{attribute 'linkalways'} 
{attribute 'no_explicit_call' := 'This FB is a CLASS and must be accessed using methods or properties'}
{attribute 'enable_dynamic_creation'}
FUNCTION_BLOCK _ETcVnKeypointDetectionTypeFAST EXTENDS EnumDatatypeBase
VAR
	localData : ETcVnKeypointDetectionTypeFAST;
	activeData : REFERENCE TO ETcVnKeypointDetectionTypeFAST;
	enumBaseDatatype : _DINT(localData);
END_VAR

METHOD PRIVATE AddLocalEnumeration
VAR_INPUT
	Enumeration : T_MAXSTRING;
	Value : ETcVnKeypointDetectionTypeFAST;
END_VAR
AddEnumeration(Enumeration, Value);
END_METHOD

PROPERTY PUBLIC Address : PVOID
GET
Address := ADR(activeData);
END_GET
END_PROPERTY

METHOD PUBLIC ClearReference
VAR_INPUT
END_VAR
activeData REF= localData;
SetBaseDatatypeReference();
END_METHOD

METHOD PUBLIC Clone : I_Datatype
VAR
    pClone : POINTER TO _ETcVnKeypointDetectionTypeFAST;
END_VAR
pClone := __NEW(_ETcVnKeypointDetectionTypeFAST(InitialValue := Value));
Clone := pClone^;
END_METHOD

METHOD FB_init : BOOL
VAR_INPUT
	bInitRetains : BOOL; // if TRUE, the retain variables are initialized (warm start / cold start)
	bInCopyCode : BOOL;  // if TRUE, the instance afterwards gets moved into the copy code (online change)
	InitialValue : ETcVnKeypointDetectionTypeFAST;
END_VAR
localData := InitialValue;
AddBaseDatatype(enumBaseDatatype);
ClearReference();

AddLocalEnumeration('TCVN_KDT_FAST_5_8', ETcVnKeypointDetectionTypeFAST.TCVN_KDT_FAST_5_8);
AddLocalEnumeration('TCVN_KDT_FAST_7_12', ETcVnKeypointDetectionTypeFAST.TCVN_KDT_FAST_7_12);
AddLocalEnumeration('TCVN_KDT_FAST_9_16', ETcVnKeypointDetectionTypeFAST.TCVN_KDT_FAST_9_16);
END_METHOD

PROPERTY PUBLIC Identifier : T_MAXSTRING
GET
Identifier := 'ETcVnKeypointDetectionTypeFAST';
END_GET
END_PROPERTY

METHOD IsEnumeratorValueEqual : BOOL
VAR_INPUT
	Enumerator : I_KeyValueForwardEnumerator;
END_VAR
VAR
	storedValue : ETcVnKeypointDetectionTypeFAST;
END_VAR
IF NOT Enumerator.TryGet(storedValue) THEN
	RETURN;
END_IF

IsEnumeratorValueEqual := storedValue = activeData;
END_METHOD

METHOD PUBLIC MakeReferenceTo
VAR_INPUT
	ReferenceTarget : REFERENCE TO ETcVnKeypointDetectionTypeFAST;
END_VAR
activeData REF= ReferenceTarget;
SetBaseDatatypeReference();
END_METHOD

METHOD PROTECTED SetBaseDatatypeReference
VAR_INPUT
END_VAR
enumBaseDatatype.MakeReferenceTo(activeData);
END_METHOD

PROPERTY PUBLIC Size : UDINT
GET
Size := SIZEOF(activeData);
END_GET
END_PROPERTY

METHOD TryMakeReferenceTo : BOOL
VAR_INPUT
	Target : I_Datatype;
END_VAR
VAR
	targetAsEnum : I_EnumDatatype;
	pTargetData : POINTER TO ETcVnKeypointDetectionTypeFAST;
END_VAR
IF NOT Target.TryResolveAsEnumDatatype(targetAsEnum) THEN
	RETURN;
END_IF

IF targetAsEnum.Identifier <> Identifier THEN
	RETURN;
END_IF

pTargetData := Target.Address;
activeData REF= pTargetData^;
SetBaseDatatypeReference();
TryMakeReferenceTo := TRUE;
END_METHOD

PROPERTY PUBLIC Value : ETcVnKeypointDetectionTypeFAST
GET
Value := activeData;
END_GET
SET
activeData := Value;
END_SET
END_PROPERTY

END_FUNCTION_BLOCK

(* stored: Version 1.1.0.1, ProductVersion 3.1.4024.12
   POU _ETcVnKeypointDetectionTypeFAST: Id {07be448e-3997-4734-bde9-814ab5e413a9}, SpecialFunc None
   Folder Constructor: Id {b3251690-2b14-4678-ad39-5ee1e766a0e5}
   Folder Private: Id {8c62b01f-6ae4-4674-bf88-22daf8e4ed6c}
   Folder Protected: Id {5503d437-72c5-4639-b842-741c26d6405f}
   Method AddLocalEnumeration: Id {20e35be3-0da7-4e45-99ec-b201ce8dc218}
   Property Address: Id {207dd583-53da-4de8-a1db-fd3bb2341452}
   Get Get: Id {6151c2e2-8467-4581-8855-ad5c272a4ded}
   Method ClearReference: Id {82950de0-52af-4252-b777-53303b1c47ca}
   Method Clone: Id {4e0f6b73-b1c6-4784-ad53-126b7ccf9759}
   Method FB_init: Id {8523375e-f772-4955-9b01-27318fa68884}
   Property Identifier: Id {4e9599ce-5bc3-4242-b903-4dd70959f735}
   Get Get: Id {ad89b73b-14c5-40cd-be12-7aec39f0f371}
   Method IsEnumeratorValueEqual: Id {481f30b9-7b77-46e5-8b15-1b6270447781}
   Method MakeReferenceTo: Id {ae3eb59f-6ea7-4eb5-be50-5db92e192155}
   Method SetBaseDatatypeReference: Id {8a7f7bb7-d680-4ce7-8372-87378f4f7d0d}
   Property Size: Id {d9ee322a-2e54-401f-80c0-31e4a8253080}
   Get Get: Id {48221eeb-6f2a-4c94-b6f0-9b43ff868869}
   Method TryMakeReferenceTo: Id {38fa76a1-03fa-4735-af08-80e0d4347368}
   Property Value: Id {1c686c5b-8c51-43e1-9771-0578e9194f49}
   Get Get: Id {34cf9d10-8949-482f-9eda-4e7216f0d1b3}
   Set Set: Id {3c4660f8-0238-4d3f-a674-4b5bf7887cf6} *)
